(* IEC 61131-3 sources: volt/packages/volt-lsp-iec/test-corpus/lenze-mid/Device/Plc Logic/Application/Library Manager/CAA Memory, 41 files *)

(* ---- VERSIONCONSTANTS.gvl ---- *)
VAR_GLOBAL
	GC_BYVERSION : BYTE := 1;
	GC_VERSION_1 : BYTE := 0;
END_VAR

(* ---- COMPARE.pou ---- *)
FUNCTION COMPARE : UINT
VAR_INPUT
	PMEMORYBLOCKA : POINTER TO BYTE;
	PMEMORYBLOCKB : POINTER TO BYTE;
	UINUMBEROFBYTES : UINT;
END_VAR
END_FUNCTION

(* ---- CRC16_CCITT.pou ---- *)
FUNCTION CRC16_CCITT : WORD
VAR_INPUT
	PMEMORYBLOCK : POINTER TO BYTE;
	UILENGTH : UINT;
END_VAR
END_FUNCTION

(* ---- CRC16_GENERIC.pou ---- *)
FUNCTION CRC16_GENERIC : WORD
VAR_INPUT
	PMEMORYBLOCK : POINTER TO BYTE;
	UILENGTH : UINT;
	WCRCINIT : WORD;
	WPOLY : WORD;
	XREFLECTINPUT : BOOL;
	XREFLECTOUTPUT : BOOL;
	WXOROUT : WORD;
END_VAR
END_FUNCTION

(* ---- CRC16_MODBUS.pou ---- *)
FUNCTION CRC16_MODBUS : WORD
VAR_INPUT
	PMEMORYBLOCK : POINTER TO BYTE;
	UILENGTH : UINT;
END_VAR
END_FUNCTION

(* ---- CRC16_STANDARD.pou ---- *)
FUNCTION CRC16_STANDARD : WORD
VAR_INPUT
	PMEMORYBLOCK : POINTER TO BYTE;
	UILENGTH : UINT;
END_VAR
END_FUNCTION

(* ---- CRC32.pou ---- *)
FUNCTION CRC32 : DWORD
VAR_INPUT
	PMEMORYBLOCK : POINTER TO BYTE;
	UILENGTH : UINT;
END_VAR
END_FUNCTION

(* ---- DECODE.pou ---- *)
FUNCTION DECODE : BOOL
VAR_INPUT
	PSOURCE : POINTER TO ARRAY [0..0] OF BYTE;
	PDESTINATION : POINTER TO ARRAY [0..0] OF DWORD;
	UINUMBEROFBYTES : UINT;
END_VAR
END_FUNCTION

(* ---- ENCODE.pou ---- *)
FUNCTION ENCODE : BOOL
VAR_INPUT
	PSOURCE : POINTER TO ARRAY [0..0] OF DWORD;
	PDESTINATION : POINTER TO ARRAY [0..0] OF BYTE;
	UINUMBEROFBYTES : UINT;
END_VAR
END_FUNCTION

(* ---- FINDBLOCK.pou ---- *)
FUNCTION FINDBLOCK : UINT
VAR_INPUT
	PMEMORYBLOCKA : POINTER TO BYTE;
	UILENGTHBLOCKA : UINT;
	PMEMORYBLOCKB : POINTER TO BYTE;
	UILENGTHBLOCKB : UINT;
END_VAR
END_FUNCTION

(* ---- FINDBYTE.pou ---- *)
FUNCTION FINDBYTE : UINT
VAR_INPUT
	PMEMORYBLOCK : POINTER TO BYTE;
	UILENGTH : UINT;
	BYVALUE : BYTE;
END_VAR
END_FUNCTION

(* ---- GETSUPPLIERVERSION.pou ---- *)
FUNCTION GETSUPPLIERVERSION : WORD
VAR_INPUT
	XDUMMY : BOOL;
END_VAR
END_FUNCTION

(* ---- HIGHBYTE.pou ---- *)
FUNCTION HIGHBYTE : BYTE
VAR_INPUT
	WVALUE : WORD;
END_VAR
END_FUNCTION

(* ---- HIGHWORD.pou ---- *)
FUNCTION HIGHWORD : WORD
VAR_INPUT
	DWVALUE : DWORD;
END_VAR
END_FUNCTION

(* ---- LOWBYTE.pou ---- *)
FUNCTION LOWBYTE : BYTE
VAR_INPUT
	WVALUE : WORD;
END_VAR
END_FUNCTION

(* ---- LOWWORD.pou ---- *)
FUNCTION LOWWORD : WORD
VAR_INPUT
	DWVALUE : DWORD;
END_VAR
END_FUNCTION

(* ---- MD5_FF.pou ---- *)
FUNCTION MD5_FF : DWORD
VAR_INPUT
	DWA : DWORD;
	DWB : DWORD;
	DWC : DWORD;
	DWD : DWORD;
	DWX : DWORD;
	DWS : UINT;
	DWT : DWORD;
END_VAR
END_FUNCTION

(* ---- MD5_GG.pou ---- *)
FUNCTION MD5_GG : DWORD
VAR_INPUT
	DWA : DWORD;
	DWB : DWORD;
	DWC : DWORD;
	DWD : DWORD;
	DWX : DWORD;
	DWS : UINT;
	DWT : DWORD;
END_VAR
END_FUNCTION

(* ---- MD5_HH.pou ---- *)
FUNCTION MD5_HH : DWORD
VAR_INPUT
	DWA : DWORD;
	DWB : DWORD;
	DWC : DWORD;
	DWD : DWORD;
	DWX : DWORD;
	DWS : UINT;
	DWT : DWORD;
END_VAR
END_FUNCTION

(* ---- MD5_II.pou ---- *)
FUNCTION MD5_II : DWORD
VAR_INPUT
	DWA : DWORD;
	DWB : DWORD;
	DWC : DWORD;
	DWD : DWORD;
	DWX : DWORD;
	DWS : UINT;
	DWT : DWORD;
END_VAR
END_FUNCTION

(* ---- MD5_TRANSFORM.pou ---- *)
FUNCTION MD5_TRANSFORM : BOOL
VAR_INPUT
	PADWSTATE : POINTER TO ARRAY [0..3] OF DWORD;
	PBUFFER : POINTER TO BYTE;
END_VAR
END_FUNCTION

(* ---- MEMFILL.pou ---- *)
FUNCTION MEMFILL : BOOL
VAR_INPUT
	PMEMORYBLOCK : POINTER TO BYTE;
	UILENGTH : UINT;
	BYFILLVALUE : BYTE;
END_VAR
END_FUNCTION

(* ---- MEMMOVE.pou ---- *)
FUNCTION MEMMOVE : BOOL
VAR_INPUT
	PSOURCE : POINTER TO BYTE;
	PDESTINATION : POINTER TO BYTE;
	UINUMBEROFBYTES : UINT;
END_VAR
END_FUNCTION

(* ---- PACKARRAYOFBOOLTOARRAYOFBYTE.pou ---- *)
FUNCTION PACKARRAYOFBOOLTOARRAYOFBYTE : UINT
VAR_INPUT
	PAXSOURCE : POINTER TO BYTE;
	PABYDESTINATION : POINTER TO BYTE;
	UINUMBEROFBITS : UINT;
END_VAR
END_FUNCTION

(* ---- PACKBITSTOBYTE.pou ---- *)
FUNCTION PACKBITSTOBYTE : BYTE
VAR_INPUT
	XBIT7 : BOOL;
	XBIT6 : BOOL;
	XBIT5 : BOOL;
	XBIT4 : BOOL;
	XBIT3 : BOOL;
	XBIT2 : BOOL;
	XBIT1 : BOOL;
	XBIT0 : BOOL;
END_VAR
END_FUNCTION

(* ---- PACKBITSTODWORD.pou ---- *)
FUNCTION PACKBITSTODWORD : DWORD
VAR_INPUT
	XBIT31 : BOOL;
	XBIT30 : BOOL;
	XBIT29 : BOOL;
	XBIT28 : BOOL;
	XBIT27 : BOOL;
	XBIT26 : BOOL;
	XBIT25 : BOOL;
	XBIT24 : BOOL;
	XBIT23 : BOOL;
	XBIT22 : BOOL;
	XBIT21 : BOOL;
	XBIT20 : BOOL;
	XBIT19 : BOOL;
	XBIT18 : BOOL;
	XBIT17 : BOOL;
	XBIT16 : BOOL;
	XBIT15 : BOOL;
	XBIT14 : BOOL;
	XBIT13 : BOOL;
	XBIT12 : BOOL;
	XBIT11 : BOOL;
	XBIT10 : BOOL;
	XBIT9 : BOOL;
	XBIT8 : BOOL;
	XBIT7 : BOOL;
	XBIT6 : BOOL;
	XBIT5 : BOOL;
	XBIT4 : BOOL;
	XBIT3 : BOOL;
	XBIT2 : BOOL;
	XBIT1 : BOOL;
	XBIT0 : BOOL;
END_VAR
END_FUNCTION

(* ---- PACKBITSTOWORD.pou ---- *)
FUNCTION PACKBITSTOWORD : WORD
VAR_INPUT
	XBIT15 : BOOL;
	XBIT14 : BOOL;
	XBIT13 : BOOL;
	XBIT12 : BOOL;
	XBIT11 : BOOL;
	XBIT10 : BOOL;
	XBIT9 : BOOL;
	XBIT8 : BOOL;
	XBIT7 : BOOL;
	XBIT6 : BOOL;
	XBIT5 : BOOL;
	XBIT4 : BOOL;
	XBIT3 : BOOL;
	XBIT2 : BOOL;
	XBIT1 : BOOL;
	XBIT0 : BOOL;
END_VAR
END_FUNCTION

(* ---- PACKBYTESTODWORD.pou ---- *)
FUNCTION PACKBYTESTODWORD : DWORD
VAR_INPUT
	BYHHBYTE : BYTE;
	BYHLBYTE : BYTE;
	BYLHBYTE : BYTE;
	BYLLBYTE : BYTE;
END_VAR
END_FUNCTION

(* ---- PACKBYTESTOWORD.pou ---- *)
FUNCTION PACKBYTESTOWORD : WORD
VAR_INPUT
	BYHIGHBYTE : BYTE;
	BYLOWBYTE : BYTE;
END_VAR
END_FUNCTION

(* ---- PACKWORDSTODWORD.pou ---- *)
FUNCTION PACKWORDSTODWORD : DWORD
VAR_INPUT
	WHIGHWORD : WORD;
	WLOWWORD : WORD;
END_VAR
END_FUNCTION

(* ---- REVERSEBITSINBYTE.pou ---- *)
FUNCTION REVERSEBITSINBYTE : BYTE
VAR_INPUT
	BYINPUT : BYTE;
END_VAR
END_FUNCTION

(* ---- REVERSEBITSINDWORD.pou ---- *)
FUNCTION REVERSEBITSINDWORD : DWORD
VAR_INPUT
	DWINPUT : DWORD;
END_VAR
END_FUNCTION

(* ---- REVERSEBITSINWORD.pou ---- *)
FUNCTION REVERSEBITSINWORD : WORD
VAR_INPUT
	WINPUT : WORD;
END_VAR
END_FUNCTION

(* ---- REVERSEBYTESINDWORD.pou ---- *)
FUNCTION REVERSEBYTESINDWORD : DWORD
VAR_INPUT
	DWINPUT : DWORD;
END_VAR
END_FUNCTION

(* ---- REVERSEBYTESINWORD.pou ---- *)
FUNCTION REVERSEBYTESINWORD : WORD
VAR_INPUT
	WINPUT : WORD;
END_VAR
END_FUNCTION

(* ---- REVERSEWORDSINDWORD.pou ---- *)
FUNCTION REVERSEWORDSINDWORD : DWORD
VAR_INPUT
	DWINPUT : DWORD;
END_VAR
END_FUNCTION

(* ---- UNPACKARRAYOFBYTE.pou ---- *)
FUNCTION UNPACKARRAYOFBYTE : UINT
VAR_INPUT
	PABYSOURCE : POINTER TO BYTE;
	PAXDESTINATION : POINTER TO BYTE;
	UINUMBEROFBITS : UINT;
END_VAR
END_FUNCTION

(* ---- MD5.pou ---- *)
FUNCTION_BLOCK MD5
VAR_INPUT
	XEXECUTE : BOOL;
	PMEMORYBLOCK : POINTER TO BYTE;
	UDINUMBEROFBYTES : UDINT;
END_VAR
VAR_OUTPUT
	XDONE : BOOL;
	XBUSY : BOOL;
	ABYDIGEST : ARRAY [0..15] OF BYTE;
END_VAR
VAR
	UDINUMBEROFBYTEPERSEGMENT : UDINT := 64;
	XEXECUTEOLD : BOOL;
	UISTEP : UINT;
	UDINUMBEROFBYTESTOTAL : UDINT;
	UILOOP : UINT;
	UDINUMBEROFBYTESUPDATED : UDINT;
	UINUMBEROFSEGMENTS : UINT;
	ADWSTATE : ARRAY [0..3] OF DWORD;
	ADWCOUNT : ARRAY [0..1] OF DWORD;
	ABYBUFFER : ARRAY [0..63] OF BYTE;
	PINPUT : POINTER TO BYTE;
	UDILENGTH : UDINT;
	UDIINDEX : UDINT;
	UDIPARTLEN : UDINT;
	UDIINPUTOFFSET : UDINT;
	INDEX : UDINT;
	PADLEN : UDINT;
	ABYBITS : ARRAY [0..7] OF BYTE;
	ABYPADDING : ARRAY [0..63] OF BYTE := [1(BYTE#16#80)];
END_VAR
END_FUNCTION_BLOCK

METHOD FINALE
END_METHOD

METHOD UPDATE
END_METHOD

METHOD INIT
END_METHOD

(* ---- UNPACKBYTE.pou ---- *)
FUNCTION_BLOCK UNPACKBYTE
VAR_INPUT
	BYVALUE : BYTE;
END_VAR
VAR_OUTPUT
	XBIT0 : BOOL;
	XBIT1 : BOOL;
	XBIT2 : BOOL;
	XBIT3 : BOOL;
	XBIT4 : BOOL;
	XBIT5 : BOOL;
	XBIT6 : BOOL;
	XBIT7 : BOOL;
END_VAR
END_FUNCTION_BLOCK

(* ---- UNPACKDWORD.pou ---- *)
FUNCTION_BLOCK UNPACKDWORD
VAR_INPUT
	DWVALUE : DWORD;
END_VAR
VAR_OUTPUT
	WLOWWORD : WORD;
	WHIGHWORD : WORD;
	BYLLBYTE : BYTE;
	BYLHBYTE : BYTE;
	BYHLBYTE : BYTE;
	BYHHBYTE : BYTE;
	XBIT0 : BOOL;
	XBIT1 : BOOL;
	XBIT2 : BOOL;
	XBIT3 : BOOL;
	XBIT4 : BOOL;
	XBIT5 : BOOL;
	XBIT6 : BOOL;
	XBIT7 : BOOL;
	XBIT8 : BOOL;
	XBIT9 : BOOL;
	XBIT10 : BOOL;
	XBIT11 : BOOL;
	XBIT12 : BOOL;
	XBIT13 : BOOL;
	XBIT14 : BOOL;
	XBIT15 : BOOL;
	XBIT16 : BOOL;
	XBIT17 : BOOL;
	XBIT18 : BOOL;
	XBIT19 : BOOL;
	XBIT20 : BOOL;
	XBIT21 : BOOL;
	XBIT22 : BOOL;
	XBIT23 : BOOL;
	XBIT24 : BOOL;
	XBIT25 : BOOL;
	XBIT26 : BOOL;
	XBIT27 : BOOL;
	XBIT28 : BOOL;
	XBIT29 : BOOL;
	XBIT30 : BOOL;
	XBIT31 : BOOL;
END_VAR
END_FUNCTION_BLOCK

(* ---- UNPACKWORD.pou ---- *)
FUNCTION_BLOCK UNPACKWORD
VAR_INPUT
	WVALUE : WORD;
END_VAR
VAR_OUTPUT
	BYLOWBYTE : BYTE;
	BYHIGHBYTE : BYTE;
	XBIT0 : BOOL;
	XBIT1 : BOOL;
	XBIT2 : BOOL;
	XBIT3 : BOOL;
	XBIT4 : BOOL;
	XBIT5 : BOOL;
	XBIT6 : BOOL;
	XBIT7 : BOOL;
	XBIT8 : BOOL;
	XBIT9 : BOOL;
	XBIT10 : BOOL;
	XBIT11 : BOOL;
	XBIT12 : BOOL;
	XBIT13 : BOOL;
	XBIT14 : BOOL;
	XBIT15 : BOOL;
END_VAR
END_FUNCTION_BLOCK
